RoboDK station: KUKAKRC2103.rdk

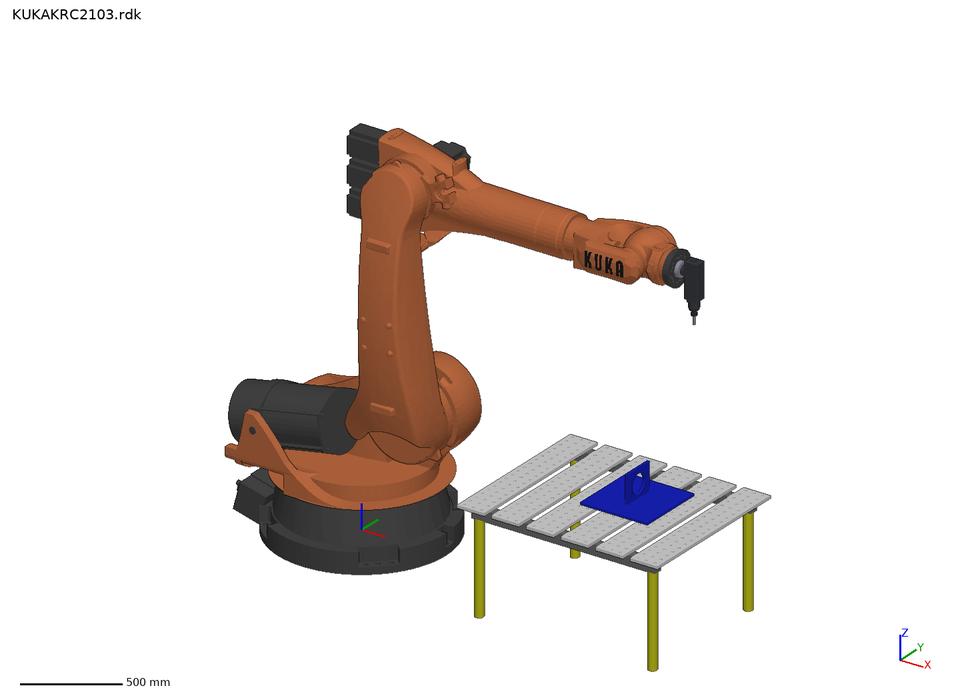
[picture v0: the station drawn from its stored meshes, robots at their saved joint values, targets as dots, program paths as lines]
Station KUKAKRC2103. Poses are relative to the parent item; angles as X-Y-Z fixed-axis rotations.
  - object Table at (1500, 0, 600) mm, size 1193.8 x 965.2 x 609.6 mm, geometry from welding_table.sld
  - frame KUKA KR 210 L180-2 Base at (0, 0, 0) mm
    - robot KUKA KR 210 L180-2: 6 axes
        modified DH rows (alpha deg, a mm, theta deg, d mm): 0, 0, 0, 750; -90, 350, 0, 0; 0, 1250, -90, 0; -90, -55, 0, 1300; 90, 0, 0, 0; -90, 0, 180, 230
        joint limits [-185, -146, -119, -350, -125, -350] to [185, 0, 155, 350, 125, 350]; home [0, -90, 90, 0, 0, 0]; saved at [0, -89.542, 89.54, 0, 0.002, 0]
      - tool Spindle, TCP at (278.6, 0, 88) mm, rotated rx 0 ry 90 rz 0 deg, size 85 x 346.5 x 128 mm
  - object Part1 at (-600, 0, -10) mm, size 400 x 400 x 176.8 mm, geometry from Part1.fbx
